(*======================================================================================================================================*)
(*RS485_COM_PRG: Beispielhaftes Programm zum Steuern von HAus-Bus.de Komponenten über RS485 mit TwinCAT
					Achtung dieser POU muss als 1ms Task Aufgerufen werden um Ordnungsgemäß zu laufen *)
(*
Date          	| Version    	| created under        	| Author          	| Remark *)
(*====================================================================================================================================================*)
(*15/05/2025   	| 1.00      		| TC3		  		| N.Kersting       | first release *)
(*====================================================================================================================================================*)

PROGRAM RS485_COM_PRG_1
VAR  
     i,h,j						:INT;
	
	fbRS485Startup				:fb_RS485Startup;		(* Startup Parametrierung der Klemme/ RS485 Bus *)
	fbRS485SendCmdFiFo			:fb_RS485FiFoMaster;	(* Sende und Empfangs FiFo für RS485 *)
	fbLineControl 				:SerialLineControl;		(* Hält die Serielle Kommunikation Aufrecht *)
	
	fComBufferReset				:ClearComBuffer;		(* Löschen des SPS Internen Bufferinhalts *)
	
	rxBuffer 					:ComBuffer;				(* COM Buffer Empfangen *)
    txBuffer 					:ComBuffer;				(* COM Buffer Senden *)
	
	
	
END_VAR

(* IDs Setzen *)
ac00_HausBusIdRS485COM();
(* RS485 Klemmen Config *)
ac01_StartupRS485COM();

ACTION ac00_HausBusIdRS485COM:
(* Initialisierung der Gerätenamen *)
(* Achtung nur Beispiele *)
fbTasterHB6F[1].I_stInput.sName := 		'Wohnzimmer';		(* Name, wie der Teilnehmer heißt / Bezeichnung *)
fbTasterHB6F[1].I_stInput.diID := 		5256;				(* Haus-Bus ID, welche auf dem Aufkleber steht  *)
		
fbTasterHB6F[2].I_stInput.sName := 		'Test1';
fbTasterHB6F[2].I_stInput.diID := 		5269;

fbTasterHB6F[3].I_stInput.sName := 		'Test2';
fbTasterHB6F[3].I_stInput.diID := 		1234;

fbTasterHB6F[4].I_stInput.sName := 		'Test3';
fbTasterHB6F[4].I_stInput.diID := 		3333;

fbTasterHB6F[5].I_stInput.sName := 		'Test4';
fbTasterHB6F[5].I_stInput.diID := 		4444;

fbTasterHB6F[6].I_stInput.sName := 		'Test5';
fbTasterHB6F[6].I_stInput.diID := 		5555;

fbTasterHB6F[7].I_stInput.sName := 		'Test6';
fbTasterHB6F[7].I_stInput.diID := 		6666;

fbTasterHB6F[8].I_stInput.sName := 		'Test7';
fbTasterHB6F[8].I_stInput.diID := 		7777;

fbTasterHB6F[9].I_stInput.sName := 		'Test8';
fbTasterHB6F[9].I_stInput.diID := 		8888;

fbTasterHB6F[10].I_stInput.sName := 	'Test9';
fbTasterHB6F[10].I_stInput.diID := 		9898;

fbRelaisHB16F[11].I_stInput.sName := 	'Jalousie 1';
fbRelaisHB16F[11].I_stInput.diID :=		5614;

fbCYDHB6F[13].I_stInput.sName :=		'CYD Test';
fbCYDHB6F[13].I_stInput.diID := 		5999;
END_ACTION

ACTION ac01_StartupRS485COM:

(* Klemmen Startup, inkl Klemmenkonfiguration usw. *)
fbRS485Startup(
	I_bExecute:= 		TRUE, 
	I_bBusOK:= 			uiEtherCATStateBK1120_RS485COM = 8
						AND uiKBusStateBK1120_RS485COM = 0, 
	I_tStartupVerz:= 	T#5S, 
	IQ_InData:= 		KL6041In, 
	IQ_OutData:= 		KL6041Out, 
	Q_sState=> , 
	Q_bStartupDone=> , 
	Q_bError=> );

(* Aktivierung der Linecontrole erst wenn Startup erfolgt *)	
IF fbRS485Startup.Q_bStartupDone
THEN
	fbLineControl(
		Mode := 		ComSerialLineMode_t.SERIALLINEMODE_KL6_22B_STANDARD,
		pComIn := 		ADR(KL6041In),
		pComOut := 		ADR(KL6041Out),
		SizeComIn := 	UINT_TO_INT(SIZEOF(KL6041In)),
		RxBuffer := 	rxBuffer,
		TxBuffer := 	txBuffer );
				
	(* Relais *)
	ac10_HausBusRelaisRS485COM();
	(* Taster *)
	ac10_HausBusTasterRS485COM();
	(* CYD *)
	ac10_HausBusCYDRS485COM();
	
	(* Senden FiFo *)
	fbRS485SendCmdFiFo(
		I_sSendCmdFiFo:= 		GVL_RS485FiFoSend.sSendFiFo, 
		I_bExecute:= 			TRUE, 
		I_bBusBelastungstest := ,
		I_bReset:= , 
		I_pTxBuffer:= 			ADR(txBuffer), 
		I_pRxBuffer:= 			ADR(rxBuffer), 
		Q_lrBusAuslastung=>		,
		Q_bBusy=> , 
		Q_bDone=> , 
		Q_bError=> , 
		Q_sState=> );
	
ELSE
	(* Com Buffer zum Resetten *)
	fComBufferReset(Buffer:= rxBuffer);
	fComBufferReset(Buffer:= txBuffer);
END_IF
END_ACTION

ACTION ac10_HausBusCYDRS485COM:
(* Bustaster Aufrufe *)
FOR j := cMaxBusRelais+cMaxBusTaster+2 TO cMaxBusRelais+cMaxBusTaster+cMaxCYD+1 BY 1 DO
			
	IF GVL_ServiceVisu.bCYDServiceAktiv[j]
	THEN
		fbCYDHB6F[j].I_stInput.iLED := GVL_ServiceVisu.stCYDService[j].iLED;
		fbCYDHB6F[j].I_stInput.iLEDBg := GVL_ServiceVisu.stCYDService[j].iLEDBg;
		fbCYDHB6F[j].I_stInput.iLEDExt := GVL_ServiceVisu.stCYDService[j].iLEDExt;
		fbCYDHB6F[j].I_stInput.bReset := GVL_ServiceVisu.stCYDService[j].bReset;
		fbCYDHB6F[j].I_stInput.bServiceMode := GVL_ServiceVisu.stCYDService[j].bServiceMode;
		fbCYDHB6F[j].I_stInput.bService := GVL_ServiceVisu.stCYDService[j].bService;
		fbCYDHB6F[j].I_stInput.bWifi := GVL_ServiceVisu.stCYDService[j].bWifi;
		fbCYDHB6F[j].I_stInput.bWebServer := GVL_ServiceVisu.stCYDService[j].bWebServer;
		
	END_IF
	
	stCYDService[j].sName :=	fbCYDHB6F[j].I_stInput.sName;
	stCYDService[j].diID :=		fbCYDHB6F[j].I_stInput.diID;
	
	fbCYDHB6F[j].I_stInput.bExecute := TRUE;
	fbCYDHB6F[j](
		I_FifoID :=			j,
		I_bPingStart:= 		TRUE , 	(* Taster Verzögert Pingen, damit weniger Busauslastung entsteht *)
		I_StringReceived:=	fbRS485SendCmdFiFo.Q_sReceiveString);
		
	(* Sendebefehle an FiFo Übergeben *)
	GVL_RS485FiFoSend.sSendFiFo[j] :=	fbCYDHB6F[j].Q_sFiFoSend;
END_FOR
END_ACTION

ACTION ac10_HausBusRelaisRS485COM:
(* BusRelais Aufrufe *)
FOR h := cMaxBusTaster +1 TO cMaxBusRelais+cMaxBusTaster+1 BY 1 DO (*cMaxBusTaster+1..cMaxBusRelais+cMaxBusTaster+1*)
		
	IF GVL_ServiceVisu.bRelaisServiceAktiv[h]
	THEN
		fbRelaisHB16F[h].I_stInput.bOut := stRelaisService[h].bOut;
		fbRelaisHB16F[h].I_stInput.bReset := stRelaisService[h].bReset;
	END_IF
	
	stRelaisService[h].sName :=	fbRelaisHB16F[h].I_stInput.sName;
	stRelaisService[h].diID :=	fbRelaisHB16F[h].I_stInput.diID;
	
	fbRelaisHB16F[h].I_stInput.bExecute := TRUE;
	fbRelaisHB16F[h](
		I_FifoID :=			h,
		I_bPingStart:= 		TRUE,	(* Direkt Starten *)
		I_StringReceived:=	fbRS485SendCmdFiFo.Q_sReceiveString);
		
	(* Sendebefehle an FiFo Übergeben *)
	GVL_RS485FiFoSend.sSendFiFo[h] :=	fbRelaisHB16F[h].Q_sFiFoSend;	
END_FOR
END_ACTION

ACTION ac10_HausBusTasterRS485COM:
(* Bustaster Aufrufe *)
FOR i := 1 TO cMaxBusTaster BY 1 DO
			
	IF GVL_ServiceVisu.bTasterServiceAktiv[i]
	THEN
		fbTasterHB6F[i].I_stInput.iLED := GVL_ServiceVisu.stTasterService[i].iLED;
		fbTasterHB6F[i].I_stInput.iLEDBg := GVL_ServiceVisu.stTasterService[i].iLEDBg;
		fbTasterHB6F[i].I_stInput.iLEDExt := GVL_ServiceVisu.stTasterService[i].iLEDExt;
		fbTasterHB6F[i].I_stInput.bReset := GVL_ServiceVisu.stTasterService[i].bReset;
	END_IF
	
	stTasterService[i].sName :=	fbTasterHB6F[i].I_stInput.sName;
	stTasterService[i].diID :=	fbTasterHB6F[i].I_stInput.diID;
	
	fbTasterHB6F[i].I_stInput.bExecute := TRUE;
	fbTasterHB6F[i](
		I_FifoID :=			i,
		I_bPingStart:= 		TRUE , 	(* Taster Verzögert Pingen, damit weniger Busauslastung entsteht *)
		I_StringReceived:=	fbRS485SendCmdFiFo.Q_sReceiveString);
		
	(* Sendebefehle an FiFo Übergeben *)
	GVL_RS485FiFoSend.sSendFiFo[i] :=	fbTasterHB6F[i].Q_sFiFoSend;
END_FOR
END_ACTION

END_PROGRAM

(* stored: Version 1.1.0.1, ProductVersion 3.1.4024.12
   POU RS485_COM_PRG_1: Id {2c5a6578-0a3e-4c7a-ab3c-a305e4780db1}, SpecialFunc None
   Folder Aufrufe: Id {ac2dc72a-faf4-4bf5-883c-68fc6fce6a2f}
   Action ac00_HausBusIdRS485COM: Id {8d09f934-10fb-4422-b01d-627fd1add300}
   Action ac01_StartupRS485COM: Id {d2e856ac-8572-4341-b59b-7b9e19140028}
   Action ac10_HausBusCYDRS485COM: Id {1feac4c3-8270-47f7-bbe2-dba512bcd624}
   Action ac10_HausBusRelaisRS485COM: Id {1cdc18a0-9a60-41ec-9231-03ba5cd5c19d}
   Action ac10_HausBusTasterRS485COM: Id {fd57d454-d9e3-4a24-960d-27efec7f7d5e} *)
